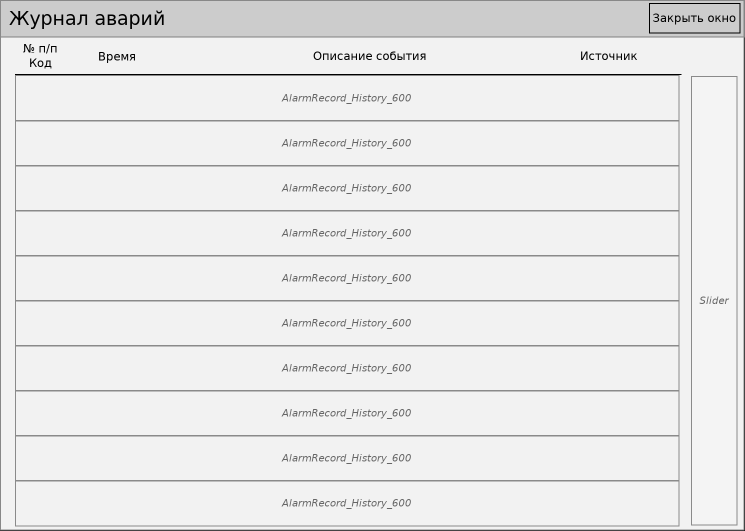
VISUALIZATION History_Of_Alarms_dialog  // 745x531
    Rectangle (0,0 745x531)
    Frame (15,75 664x46)
        shows AlarmRecord_History_600(AlarmRecord := PRG_Alarms_Core.HMI_HistoryAlarms[1], RecNum := PRG_Alarms_Core.HMI_NumsHY[1])
    Frame (15,120 664x46)
        shows AlarmRecord_History_600(AlarmRecord := PRG_Alarms_Core.HMI_HistoryAlarms[2], RecNum := PRG_Alarms_Core.HMI_NumsHY[2])
    Frame (15,165 664x46)
        shows AlarmRecord_History_600(AlarmRecord := PRG_Alarms_Core.HMI_HistoryAlarms[3], RecNum := PRG_Alarms_Core.HMI_NumsHY[3])
    Frame (15,210 664x46)
        shows AlarmRecord_History_600(AlarmRecord := PRG_Alarms_Core.HMI_HistoryAlarms[4], RecNum := PRG_Alarms_Core.HMI_NumsHY[4])
    Frame (15,255 664x46)
        shows AlarmRecord_History_600(AlarmRecord := PRG_Alarms_Core.HMI_HistoryAlarms[5], RecNum := PRG_Alarms_Core.HMI_NumsHY[5])
    Frame (15,300 664x46)
        shows AlarmRecord_History_600(AlarmRecord := PRG_Alarms_Core.HMI_HistoryAlarms[6], RecNum := PRG_Alarms_Core.HMI_NumsHY[6])
    Frame (15,345 664x46)
        shows AlarmRecord_History_600(AlarmRecord := PRG_Alarms_Core.HMI_HistoryAlarms[7], RecNum := PRG_Alarms_Core.HMI_NumsHY[7])
    Frame (15,390 664x46)
        shows AlarmRecord_History_600(AlarmRecord := PRG_Alarms_Core.HMI_HistoryAlarms[8], RecNum := PRG_Alarms_Core.HMI_NumsHY[8])
    Frame (15,435 664x46)
        shows AlarmRecord_History_600(AlarmRecord := PRG_Alarms_Core.HMI_HistoryAlarms[9], RecNum := PRG_Alarms_Core.HMI_NumsHY[9])
    Frame (15,480 664x46)
        shows AlarmRecord_History_600(AlarmRecord := PRG_Alarms_Core.HMI_HistoryAlarms[10], RecNum := PRG_Alarms_Core.HMI_NumsHY[10])
    Slider (691,76 46x449), variable: PRG_Alarms_Core.HMI_CurShiftHY, scale 0..1000
    Label (17,41 47x30), "№ п/п Код"
    Label (310,41 216x30), "Описание события"
    Label (577,41 77x30), "Источник"
    Label (91,47 52x19), "Время"
    Line (15,74) (681,74)
    Rectangle (0,0 745x37), "Журнал аварий"
    RoundedRectangle (649,3 91x30), "Закрыть окно"
        OnMouseClick: CloseDialog Dialog=History_Of_Alarms_dialog, Result=OK, NumpadKeypadSet=True
END_VISUALIZATION

(* stored: Version 1.1.0.1, ProductVersion 3.1.4024.3
   Visu History_Of_Alarms_dialog: Id {14318430-d88b-42df-9468-92f5fd8abf86} *)
